(* PLC project Unnamed, Unknown Unnamed 1 *)
(* stored: creationDateTime 2023-03-24T21:00:34, modificationDateTime 2023-03-25T07:28:05 *)

PROGRAM PL
  VAR
    START AT %IX100.0 : BOOL;
    STOP AT %IX100.1 : BOOL;
    SEN1 AT %IX100.2 : BOOL;
    SEN2 AT %IX100.3 : BOOL;
    VIR1 AT %QX0.0 : BOOL;
    VIR2 AT %QX0.1 : BOOL;
    MC1start1 AT %QX100.0 : BOOL;
    MC1stop2 AT %QX100.1 : BOOL;
    LIDS AT %QX100.2 : BOOL;
    CON AT %QX100.3 : BOOL;
  END_VAR
  VAR
    TON1 : TON;
  END_VAR

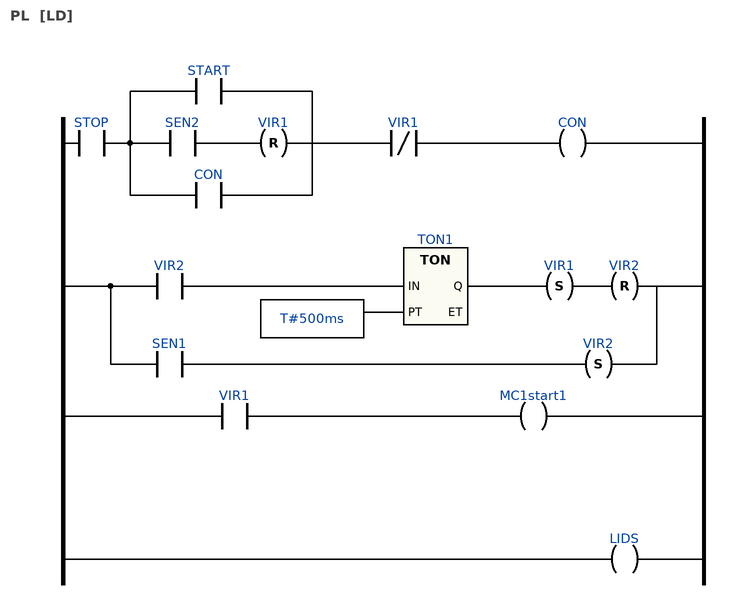
(* LD diagram, written out as Structured Text *)
IF STOP AND SEN2 THEN VIR1 := FALSE; END_IF;
CON := STOP AND (START OR CON OR SEN2) AND NOT VIR1;
TON1(IN := VIR2, PT := T#500ms);
IF TON1.Q THEN VIR1 := TRUE; END_IF;
IF TON1.Q THEN VIR2 := FALSE; END_IF;
IF SEN1 THEN VIR2 := TRUE; END_IF;
MC1start1 := VIR1;
LIDS := TRUE;
END_PROGRAM

CONFIGURATION Config0
  RESOURCE Res0 ON PLC
    TASK task0(INTERVAL := T#20ms, PRIORITY := 0);
    PROGRAM instance0 WITH task0 : PL;
  END_RESOURCE
END_CONFIGURATION
